// TIA Portal V19 export
TYPE "type_teachPara_axis"
// stored: Access Published
   STRUCT
      position : Array[0..99] of LReal;
   END_STRUCT;
END_TYPE
